PROGRAM EM06_Picking
VAR
	
	//Backbone
	FB_StateMachine_Picking			: FB_StateManager;
	bFl_RunningMachinePicking		: BOOL;
	bFl_SeqReset					: BOOL;
	bFl_Manual						: BOOL;
	CheckStatusPicking				: checkstatus;
	AlarmEventHistory				: ARRAY[1..20] OF Alarm_Event_History;
	ProductFound					: ARRAY [1..4] OF BOOL;
	
	//Motor
	Motor_BoxPicking				: MotorManagement;
	bFl_MotorPicking				: BOOL;
	Motor_Picking_Error				: BOOL;
	Motor_Picking_ErrorID			: UINT;
	
	//Pneumatic
	Pneumatic_GapMaker				: Pneumatic_2Coil_Management;
	bFl_GapMaker_Rtc				: BOOL;
	bFl_GapMaker_Adv				: BOOL;
	Pneu_GapMaker_Error				: BOOL;	
	Pneu_GapMaker_ErrorMsg			: STRING;
	
	Pneumatic_Centering				: Pneumatic_1Coil_Management;
	bFl_Centering					: BOOL;
	Pneu_Centering_Error			: BOOL;	
	Pneu_Centering_ErrorMsg			: STRING;
	
	//Picking
	Picking							: FB_Picking;
	
	//Barcode Reader
	bFl_BarcodeChecked				: BOOL;
	bFl_TriggerBarcode				: BOOL;
	bFl_DoneRead_Barcode_Picking	: ARRAY [1..4] OF BOOL;
	bFl_GoodRead_Barcode_Picking	: ARRAY [1..4] OF BOOL;
	bFl_BadRead_Barcode_Picking		: ARRAY [1..4] OF BOOL;
	BarcodeInspection				: FB_BarcodeInspection;
	BarcodeReader_Picking1			: DM_Connect;
	BarcodeReader_Picking2			: DM_Connect;
	BarcodeReader_Picking3			: DM_Connect;
	BarcodeReader_Picking4			: DM_Connect;
	DataBarcode_Picking1			: STRING;
	DataBarcode_Picking2			: STRING;
	DataBarcode_Picking3			: STRING;
	DataBarcode_Picking4			: STRING;
	Barcode1_Error					: BOOL;
	Barcode2_Error					: BOOL;
	Barcode3_Error					: BOOL;
	Barcode4_Error					: BOOL;
	TestRun							: BOOL;
	TestTrigger						: BOOL;
	LEN1							: INT;
	POS1							: INT;
	POS2							: INT;
	LEN_2							: INT;
	LinkUp							: STRING(255);
	RotatePicking					: RotatePick;
	DonePick						: BOOL;
	bFL_Safety						: BOOL;
	AutoReset						: BOOL;
	TON_Auto						: TON;
	AutoAck							: BOOL;
	AutoRun							: BOOL;
	TOF_Run							: TOF;
	TOF_Reset						: TOF;
	AlarmEventActive				: ARRAY[1..20] OF Alarm_Event_Active;
	RejectMsgList					: RejectMsgHandling;
	bReject							: BOOL;
	RejectID						: INT;
	RejectMsg						: STRING;
	CounterReject					: UINT;
	bRotate							: BOOL;
	BarcodeReader_Picking2B			: DM_Connect;
	Barcode2B_Error					: BOOL;
	DataBarcode_Picking2B			: STRING;
	bFl_DoneRead_Barcode_Picking2B	: BOOL;
	
	BarcodeReader_Picking3B			: DM_Connect;
	Barcode3B_Error					: BOOL;
	DataBarcode_Picking3B			: STRING;
	intRotatePick					: USINT;
END_VAR
VAR // added by the converter: edge detectors and wires of the graphical bodies
    _w1 : BOOL;
END_VAR

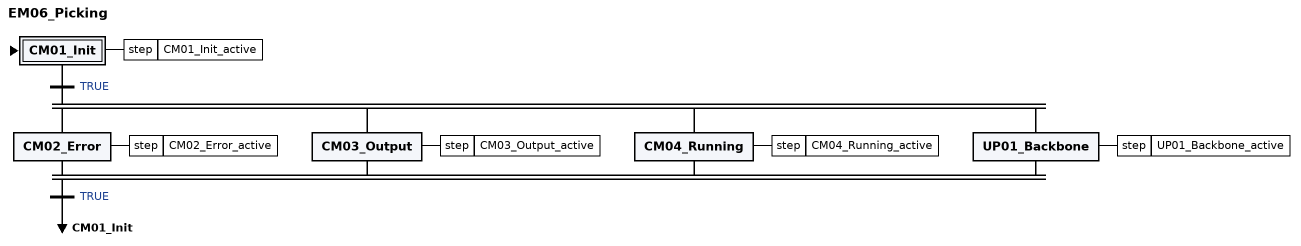
INITIAL_STEP CM01_Init:
    CM01_Init_active(N);  // step action
END_STEP
TRANSITION FROM CM01_Init TO (CM02_Error, CM03_Output, CM04_Running, UP01_Backbone)
    := TRUE;
END_TRANSITION
STEP CM02_Error:
    CM02_Error_active(N);  // step action
END_STEP
STEP CM03_Output:
    CM03_Output_active(N);  // step action
END_STEP
STEP CM04_Running:
    CM04_Running_active(N);  // step action
END_STEP
STEP UP01_Backbone:
    UP01_Backbone_active(N);  // step action
END_STEP
TRANSITION FROM (CM02_Error, CM03_Output, CM04_Running, UP01_Backbone) TO CM01_Init
    := TRUE;
END_TRANSITION

ACTION CM01_Init_active:
Data_GVL.bFL_StartPicking			:= Status_GVL.bFl_RunButton_Robotic OR HMI_GVL.bStartButtonPicking OR HMI_GVL.bAutoStartPicking;
Data_GVL.bFL_StopPicking			:= NOT Status_GVL.bFl_StopButton_Robotic OR HMI_GVL.bStopButtonPicking;
Data_GVL.bFL_ResetPicking			:= Status_GVL.bFl_ResetButton_Robotic OR HMI_GVL.bResetButtonPicking OR HMI_GVL.bAutoResetPicking;
Data_GVL.bFL_AckPicking				:= Status_GVL.bFl_Acknowledge_Robotic OR HMI_GVL.bAcknowledgeButtonPicking OR HMI_GVL.bAutoAcknowledgePicking;
Data_GVL.bFL_AutoManuaModePicking 	:= Status_GVL.bFl_Manual_Robotic OR HMI_GVL.bTestModeEnablePicking;
bFl_RunningMachinePicking			:= Data_GVL.stStateMachinePicking.Running;
bFl_Manual							:= Data_GVL.stStateMachinePicking.ManualMode;
bFl_SeqReset						:= NOT Status_GVL.bFl_EStop_Robotic;
bFL_Safety							:= Status_GVL.bFl_EStop_Robotic AND Status_GVL.bSafety_DoorRobotic AND Status_GVL.bAirPressure_Robotic;



(*=================Convert Timer============================*)
Data_GVL.Tmr_Picking	:= ConvertMilliSecTimeData(HMI_GVL.Tmr_Picking);
Data_GVL.Tmr_Centering	:= ConvertMilliSecTimeData(HMI_GVL.Tmr_Centering);

(*=================Auto Flushing============================*)
//Place1
IF ProductFound[1] AND HMI_GVL.arCountReal[1] > 1 THEN
	Status_GVL.AutoFlush_Placing1	:= TRUE;
ELSE
	Status_GVL.AutoFlush_Placing1	:= FALSE;
END_IF

//Place2
IF ProductFound[2] AND HMI_GVL.arCountReal[2] > 1 THEN
	Status_GVL.AutoFlush_Placing2	:= TRUE;
ELSE
	Status_GVL.AutoFlush_Placing2	:= FALSE;
END_IF

//Place3
IF ProductFound[3] AND HMI_GVL.arCountReal[3] > 1 THEN
	Status_GVL.AutoFlush_Placing3	:= TRUE;
ELSE
	Status_GVL.AutoFlush_Placing3	:= FALSE;
END_IF

//Place4
IF ProductFound[4] AND HMI_GVL.arCountReal[4] > 1 THEN
	Status_GVL.AutoFlush_Placing4	:= TRUE;
ELSE
	Status_GVL.AutoFlush_Placing4	:= FALSE;
END_IF
END_ACTION

ACTION CM02_Error_active:
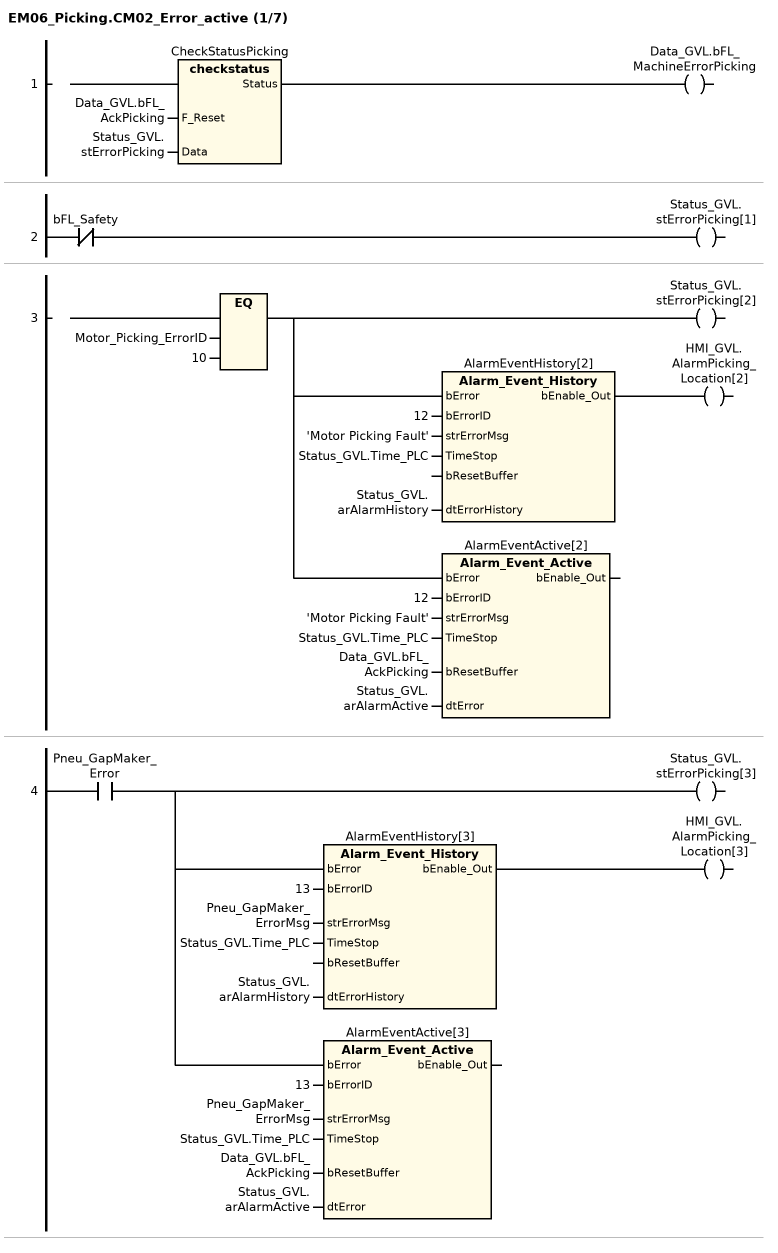
// NETWORK 1
CheckStatusPicking(F_Reset := Data_GVL.bFL_AckPicking, Data := Status_GVL.stErrorPicking); // checkstatus
Data_GVL.bFL_MachineErrorPicking := CheckStatusPicking.Status;

// NETWORK 2
Status_GVL.stErrorPicking[1] := NOT bFL_Safety;

// NETWORK 3
_w1 := Motor_Picking_ErrorID = 10;
Status_GVL.stErrorPicking[2] := _w1;
AlarmEventHistory[2](
    bError := _w1,
    bErrorID := 12,
    strErrorMsg := 'Motor Picking Fault',
    TimeStop := Status_GVL.Time_PLC,
    dtErrorHistory := Status_GVL.arAlarmHistory); // Alarm_Event_History
HMI_GVL.AlarmPicking_Location[2] := AlarmEventHistory[2].bEnable_Out;
AlarmEventActive[2](
    bError := _w1,
    bErrorID := 12,
    strErrorMsg := 'Motor Picking Fault',
    TimeStop := Status_GVL.Time_PLC,
    bResetBuffer := Data_GVL.bFL_AckPicking,
    dtError := Status_GVL.arAlarmActive); // Alarm_Event_Active

// NETWORK 4
Status_GVL.stErrorPicking[3] := Pneu_GapMaker_Error;
AlarmEventHistory[3](
    bError := Pneu_GapMaker_Error,
    bErrorID := 13,
    strErrorMsg := Pneu_GapMaker_ErrorMsg,
    TimeStop := Status_GVL.Time_PLC,
    dtErrorHistory := Status_GVL.arAlarmHistory); // Alarm_Event_History
HMI_GVL.AlarmPicking_Location[3] := AlarmEventHistory[3].bEnable_Out;
AlarmEventActive[3](
    bError := Pneu_GapMaker_Error,
    bErrorID := 13,
    strErrorMsg := Pneu_GapMaker_ErrorMsg,
    TimeStop := Status_GVL.Time_PLC,
    bResetBuffer := Data_GVL.bFL_AckPicking,
    dtError := Status_GVL.arAlarmActive); // Alarm_Event_Active

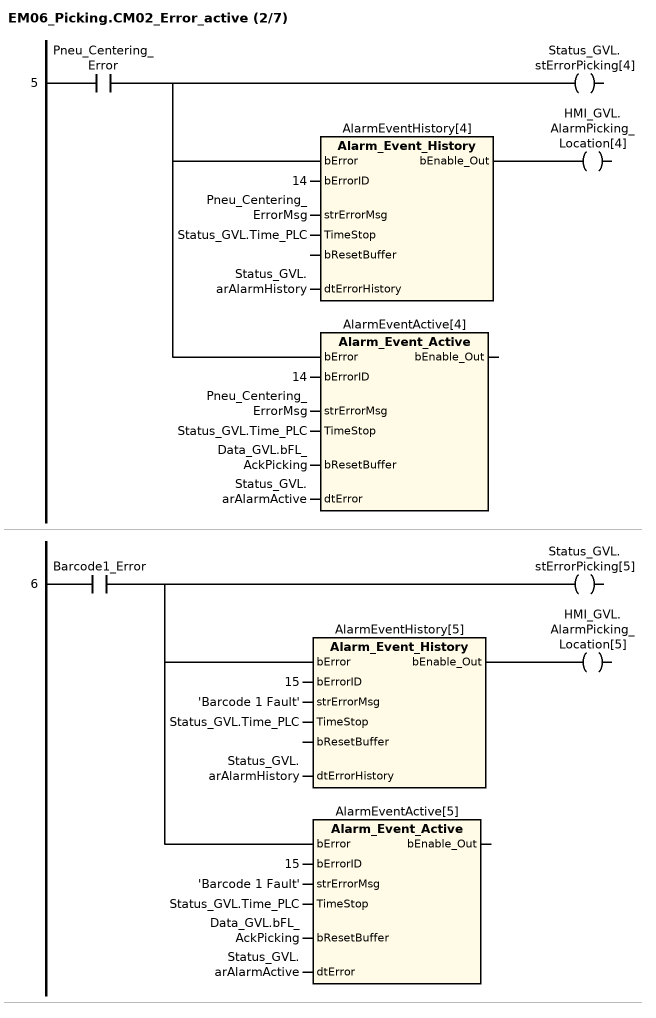
// NETWORK 5
Status_GVL.stErrorPicking[4] := Pneu_Centering_Error;
AlarmEventHistory[4](
    bError := Pneu_Centering_Error,
    bErrorID := 14,
    strErrorMsg := Pneu_Centering_ErrorMsg,
    TimeStop := Status_GVL.Time_PLC,
    dtErrorHistory := Status_GVL.arAlarmHistory); // Alarm_Event_History
HMI_GVL.AlarmPicking_Location[4] := AlarmEventHistory[4].bEnable_Out;
AlarmEventActive[4](
    bError := Pneu_Centering_Error,
    bErrorID := 14,
    strErrorMsg := Pneu_Centering_ErrorMsg,
    TimeStop := Status_GVL.Time_PLC,
    bResetBuffer := Data_GVL.bFL_AckPicking,
    dtError := Status_GVL.arAlarmActive); // Alarm_Event_Active

// NETWORK 6
Status_GVL.stErrorPicking[5] := Barcode1_Error;
AlarmEventHistory[5](
    bError := Barcode1_Error,
    bErrorID := 15,
    strErrorMsg := 'Barcode 1 Fault',
    TimeStop := Status_GVL.Time_PLC,
    dtErrorHistory := Status_GVL.arAlarmHistory); // Alarm_Event_History
HMI_GVL.AlarmPicking_Location[5] := AlarmEventHistory[5].bEnable_Out;
AlarmEventActive[5](
    bError := Barcode1_Error,
    bErrorID := 15,
    strErrorMsg := 'Barcode 1 Fault',
    TimeStop := Status_GVL.Time_PLC,
    bResetBuffer := Data_GVL.bFL_AckPicking,
    dtError := Status_GVL.arAlarmActive); // Alarm_Event_Active

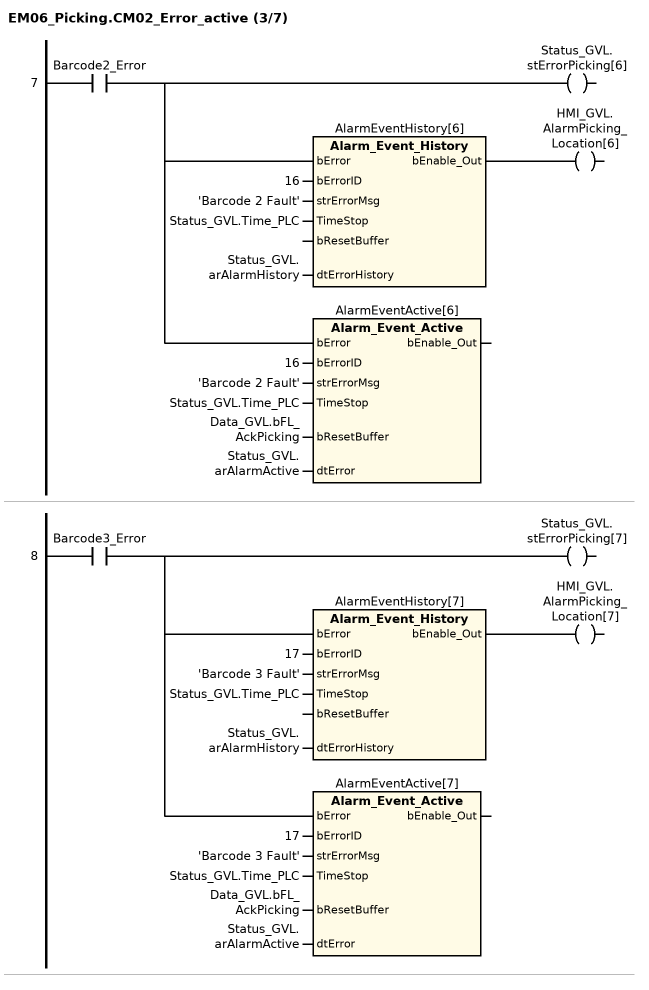
// NETWORK 7
Status_GVL.stErrorPicking[6] := Barcode2_Error;
AlarmEventHistory[6](
    bError := Barcode2_Error,
    bErrorID := 16,
    strErrorMsg := 'Barcode 2 Fault',
    TimeStop := Status_GVL.Time_PLC,
    dtErrorHistory := Status_GVL.arAlarmHistory); // Alarm_Event_History
HMI_GVL.AlarmPicking_Location[6] := AlarmEventHistory[6].bEnable_Out;
AlarmEventActive[6](
    bError := Barcode2_Error,
    bErrorID := 16,
    strErrorMsg := 'Barcode 2 Fault',
    TimeStop := Status_GVL.Time_PLC,
    bResetBuffer := Data_GVL.bFL_AckPicking,
    dtError := Status_GVL.arAlarmActive); // Alarm_Event_Active

// NETWORK 8
Status_GVL.stErrorPicking[7] := Barcode3_Error;
AlarmEventHistory[7](
    bError := Barcode3_Error,
    bErrorID := 17,
    strErrorMsg := 'Barcode 3 Fault',
    TimeStop := Status_GVL.Time_PLC,
    dtErrorHistory := Status_GVL.arAlarmHistory); // Alarm_Event_History
HMI_GVL.AlarmPicking_Location[7] := AlarmEventHistory[7].bEnable_Out;
AlarmEventActive[7](
    bError := Barcode3_Error,
    bErrorID := 17,
    strErrorMsg := 'Barcode 3 Fault',
    TimeStop := Status_GVL.Time_PLC,
    bResetBuffer := Data_GVL.bFL_AckPicking,
    dtError := Status_GVL.arAlarmActive); // Alarm_Event_Active

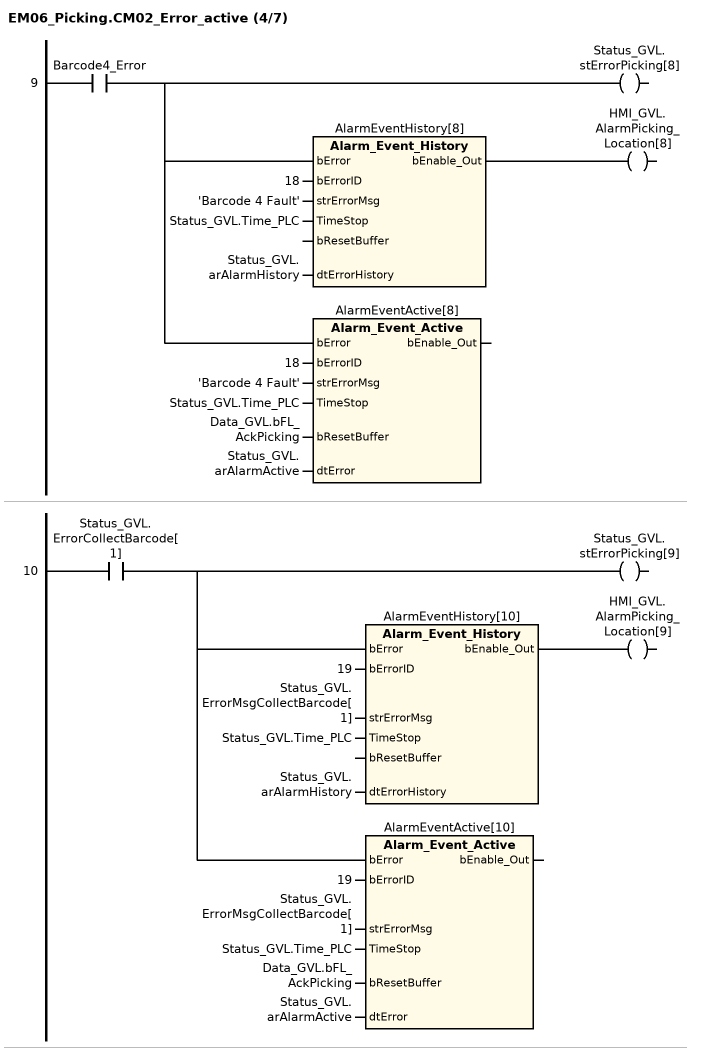
// NETWORK 9
Status_GVL.stErrorPicking[8] := Barcode4_Error;
AlarmEventHistory[8](
    bError := Barcode4_Error,
    bErrorID := 18,
    strErrorMsg := 'Barcode 4 Fault',
    TimeStop := Status_GVL.Time_PLC,
    dtErrorHistory := Status_GVL.arAlarmHistory); // Alarm_Event_History
HMI_GVL.AlarmPicking_Location[8] := AlarmEventHistory[8].bEnable_Out;
AlarmEventActive[8](
    bError := Barcode4_Error,
    bErrorID := 18,
    strErrorMsg := 'Barcode 4 Fault',
    TimeStop := Status_GVL.Time_PLC,
    bResetBuffer := Data_GVL.bFL_AckPicking,
    dtError := Status_GVL.arAlarmActive); // Alarm_Event_Active

// NETWORK 10
Status_GVL.stErrorPicking[9] := Status_GVL.ErrorCollectBarcode[1];
AlarmEventHistory[10](
    bError := Status_GVL.ErrorCollectBarcode[1],
    bErrorID := 19,
    strErrorMsg := Status_GVL.ErrorMsgCollectBarcode[1],
    TimeStop := Status_GVL.Time_PLC,
    dtErrorHistory := Status_GVL.arAlarmHistory); // Alarm_Event_History
HMI_GVL.AlarmPicking_Location[9] := AlarmEventHistory[10].bEnable_Out;
AlarmEventActive[10](
    bError := Status_GVL.ErrorCollectBarcode[1],
    bErrorID := 19,
    strErrorMsg := Status_GVL.ErrorMsgCollectBarcode[1],
    TimeStop := Status_GVL.Time_PLC,
    bResetBuffer := Data_GVL.bFL_AckPicking,
    dtError := Status_GVL.arAlarmActive); // Alarm_Event_Active

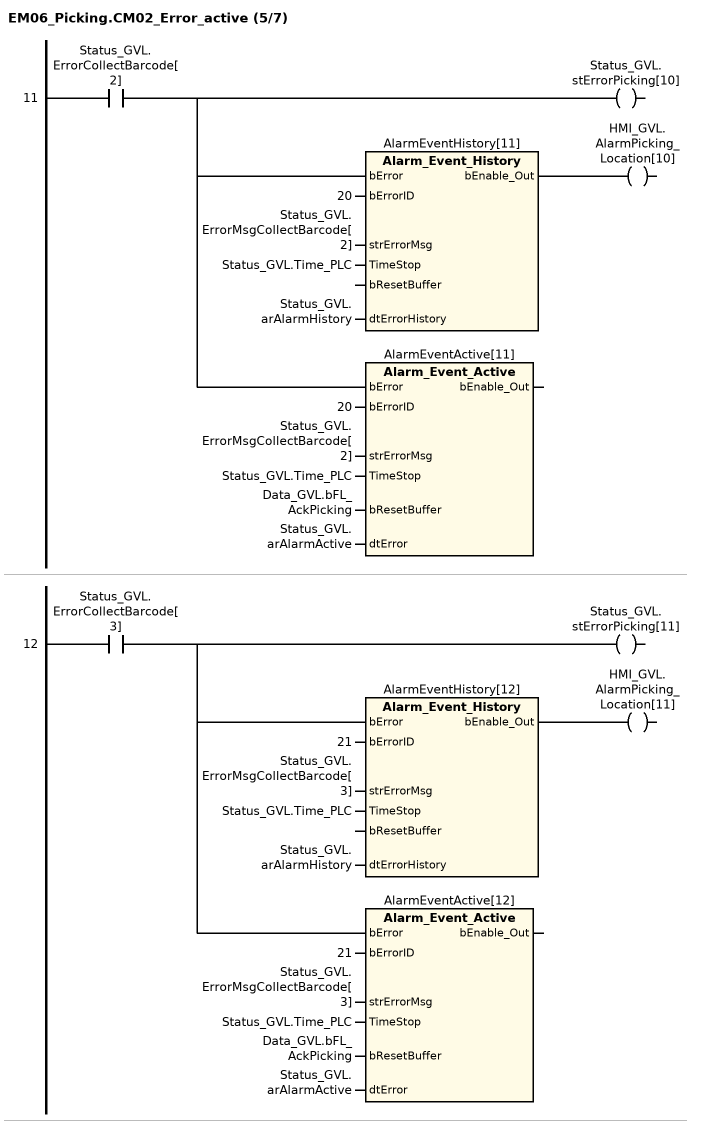
// NETWORK 11
Status_GVL.stErrorPicking[10] := Status_GVL.ErrorCollectBarcode[2];
AlarmEventHistory[11](
    bError := Status_GVL.ErrorCollectBarcode[2],
    bErrorID := 20,
    strErrorMsg := Status_GVL.ErrorMsgCollectBarcode[2],
    TimeStop := Status_GVL.Time_PLC,
    dtErrorHistory := Status_GVL.arAlarmHistory); // Alarm_Event_History
HMI_GVL.AlarmPicking_Location[10] := AlarmEventHistory[11].bEnable_Out;
AlarmEventActive[11](
    bError := Status_GVL.ErrorCollectBarcode[2],
    bErrorID := 20,
    strErrorMsg := Status_GVL.ErrorMsgCollectBarcode[2],
    TimeStop := Status_GVL.Time_PLC,
    bResetBuffer := Data_GVL.bFL_AckPicking,
    dtError := Status_GVL.arAlarmActive); // Alarm_Event_Active

// NETWORK 12
Status_GVL.stErrorPicking[11] := Status_GVL.ErrorCollectBarcode[3];
AlarmEventHistory[12](
    bError := Status_GVL.ErrorCollectBarcode[3],
    bErrorID := 21,
    strErrorMsg := Status_GVL.ErrorMsgCollectBarcode[3],
    TimeStop := Status_GVL.Time_PLC,
    dtErrorHistory := Status_GVL.arAlarmHistory); // Alarm_Event_History
HMI_GVL.AlarmPicking_Location[11] := AlarmEventHistory[12].bEnable_Out;
AlarmEventActive[12](
    bError := Status_GVL.ErrorCollectBarcode[3],
    bErrorID := 21,
    strErrorMsg := Status_GVL.ErrorMsgCollectBarcode[3],
    TimeStop := Status_GVL.Time_PLC,
    bResetBuffer := Data_GVL.bFL_AckPicking,
    dtError := Status_GVL.arAlarmActive); // Alarm_Event_Active

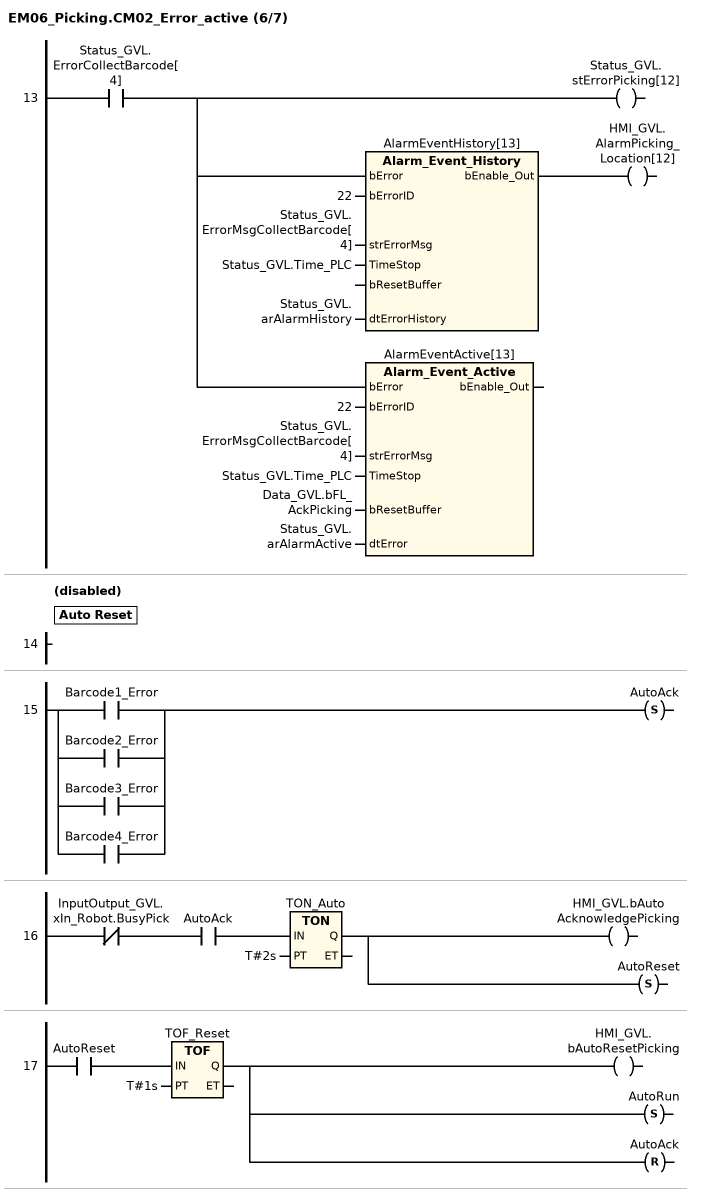
// NETWORK 13
Status_GVL.stErrorPicking[12] := Status_GVL.ErrorCollectBarcode[4];
AlarmEventHistory[13](
    bError := Status_GVL.ErrorCollectBarcode[4],
    bErrorID := 22,
    strErrorMsg := Status_GVL.ErrorMsgCollectBarcode[4],
    TimeStop := Status_GVL.Time_PLC,
    dtErrorHistory := Status_GVL.arAlarmHistory); // Alarm_Event_History
HMI_GVL.AlarmPicking_Location[12] := AlarmEventHistory[13].bEnable_Out;
AlarmEventActive[13](
    bError := Status_GVL.ErrorCollectBarcode[4],
    bErrorID := 22,
    strErrorMsg := Status_GVL.ErrorMsgCollectBarcode[4],
    TimeStop := Status_GVL.Time_PLC,
    bResetBuffer := Data_GVL.bFL_AckPicking,
    dtError := Status_GVL.arAlarmActive); // Alarm_Event_Active

// NETWORK 14 (disabled)
// label: Auto Reset

// NETWORK 15
AutoAck S= Barcode1_Error OR Barcode2_Error OR Barcode3_Error OR Barcode4_Error;

// NETWORK 16
TON_Auto(IN := NOT InputOutput_GVL.xIn_Robot.BusyPick AND AutoAck, PT := T#2s); // TON
HMI_GVL.bAutoAcknowledgePicking := TON_Auto.Q;
AutoReset S= TON_Auto.Q;

// NETWORK 17
TOF_Reset(IN := AutoReset, PT := T#1s); // TOF
HMI_GVL.bAutoResetPicking := TOF_Reset.Q;
AutoRun S= TOF_Reset.Q;
AutoAck R= TOF_Reset.Q;

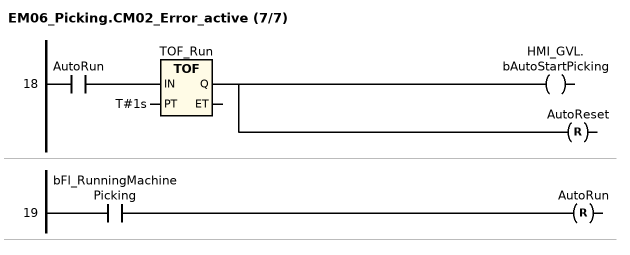
// NETWORK 18
TOF_Run(IN := AutoRun, PT := T#1s); // TOF
HMI_GVL.bAutoStartPicking := TOF_Run.Q;
AutoReset R= TOF_Run.Q;

// NETWORK 19
AutoRun R= bFl_RunningMachinePicking;
END_ACTION

ACTION CM03_Output_active:
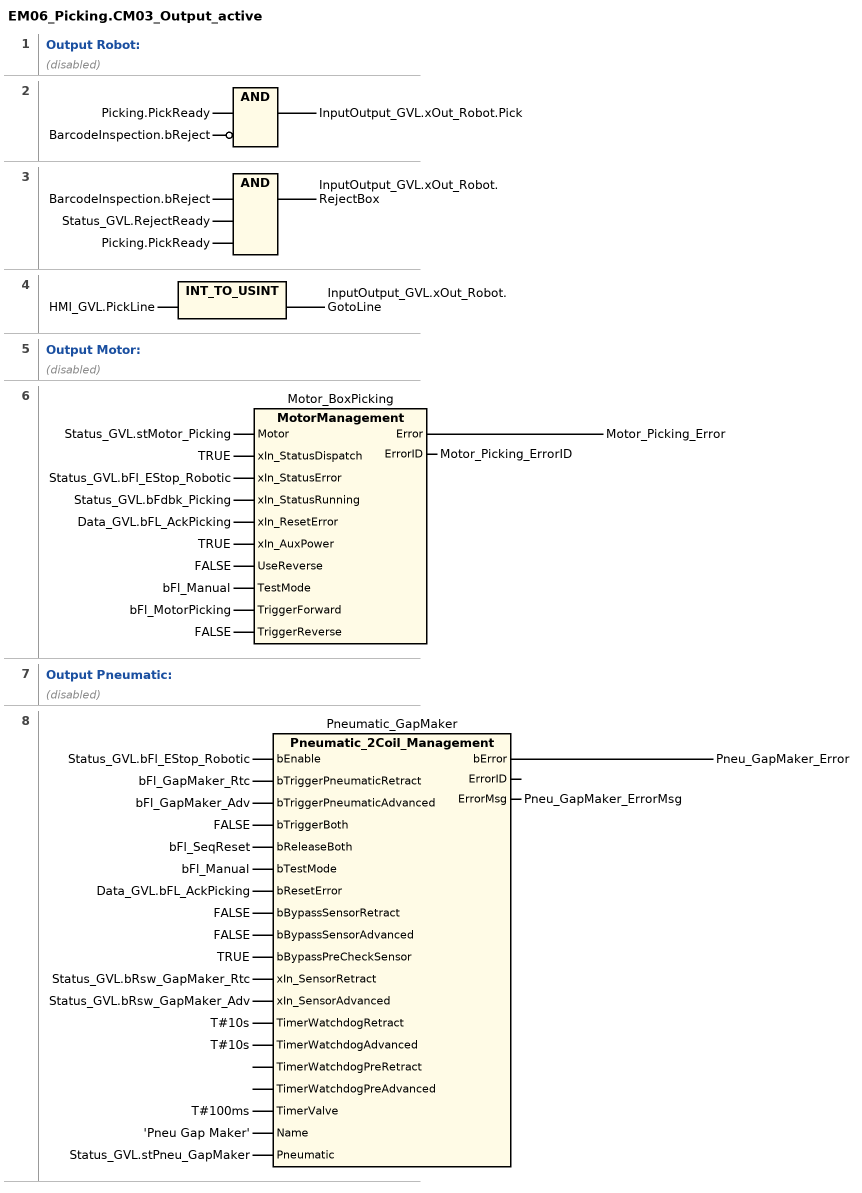
// NETWORK 1 (disabled)
// label: Output Robot

// NETWORK 2
InputOutput_GVL.xOut_Robot.Pick := Picking.PickReady AND NOT BarcodeInspection.bReject;

// NETWORK 3
InputOutput_GVL.xOut_Robot.RejectBox := BarcodeInspection.bReject AND Status_GVL.RejectReady AND Picking.PickReady;

// NETWORK 4
InputOutput_GVL.xOut_Robot.GotoLine := INT_TO_USINT(HMI_GVL.PickLine);

// NETWORK 5 (disabled)
// label: Output Motor

// NETWORK 6
Motor_BoxPicking(
    Motor := Status_GVL.stMotor_Picking,
    xIn_StatusDispatch := TRUE,
    xIn_StatusError := Status_GVL.bFl_EStop_Robotic,
    xIn_StatusRunning := Status_GVL.bFdbk_Picking,
    xIn_ResetError := Data_GVL.bFL_AckPicking,
    xIn_AuxPower := TRUE,
    UseReverse := FALSE,
    TestMode := bFl_Manual,
    TriggerForward := bFl_MotorPicking,
    TriggerReverse := FALSE,
    ErrorID => Motor_Picking_ErrorID); // MotorManagement
Motor_Picking_Error := Motor_BoxPicking.Error;

// NETWORK 7 (disabled)
// label: Output Pneumatic

// NETWORK 8
Pneumatic_GapMaker(
    bEnable := Status_GVL.bFl_EStop_Robotic,
    bTriggerPneumaticRetract := bFl_GapMaker_Rtc,
    bTriggerPneumaticAdvanced := bFl_GapMaker_Adv,
    bTriggerBoth := FALSE,
    bReleaseBoth := bFl_SeqReset,
    bTestMode := bFl_Manual,
    bResetError := Data_GVL.bFL_AckPicking,
    bBypassSensorRetract := FALSE,
    bBypassSensorAdvanced := FALSE,
    bBypassPreCheckSensor := TRUE,
    xIn_SensorRetract := Status_GVL.bRsw_GapMaker_Rtc,
    xIn_SensorAdvanced := Status_GVL.bRsw_GapMaker_Adv,
    TimerWatchdogRetract := T#10s,
    TimerWatchdogAdvanced := T#10s,
    TimerValve := T#100ms,
    Name := 'Pneu Gap Maker',
    Pneumatic := Status_GVL.stPneu_GapMaker,
    ErrorMsg => Pneu_GapMaker_ErrorMsg); // Pneumatic_2Coil_Management
Pneu_GapMaker_Error := Pneumatic_GapMaker.bError;

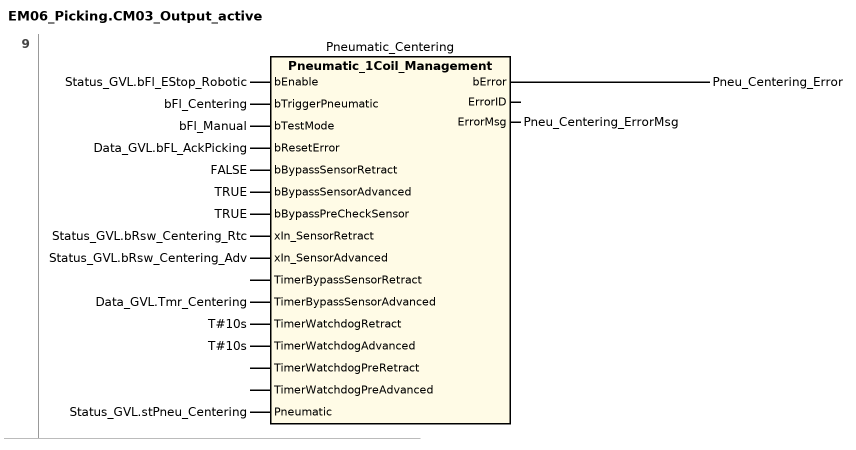
// NETWORK 9
Pneumatic_Centering(
    bEnable := Status_GVL.bFl_EStop_Robotic,
    bTriggerPneumatic := bFl_Centering,
    bTestMode := bFl_Manual,
    bResetError := Data_GVL.bFL_AckPicking,
    bBypassSensorRetract := FALSE,
    bBypassSensorAdvanced := TRUE,
    bBypassPreCheckSensor := TRUE,
    xIn_SensorRetract := Status_GVL.bRsw_Centering_Rtc,
    xIn_SensorAdvanced := Status_GVL.bRsw_Centering_Adv,
    TimerBypassSensorAdvanced := Data_GVL.Tmr_Centering,
    TimerWatchdogRetract := T#10s,
    TimerWatchdogAdvanced := T#10s,
    Pneumatic := Status_GVL.stPneu_Centering,
    ErrorMsg => Pneu_Centering_ErrorMsg); // Pneumatic_1Coil_Management
Pneu_Centering_Error := Pneumatic_Centering.bError;
END_ACTION

ACTION CM04_Running_active:
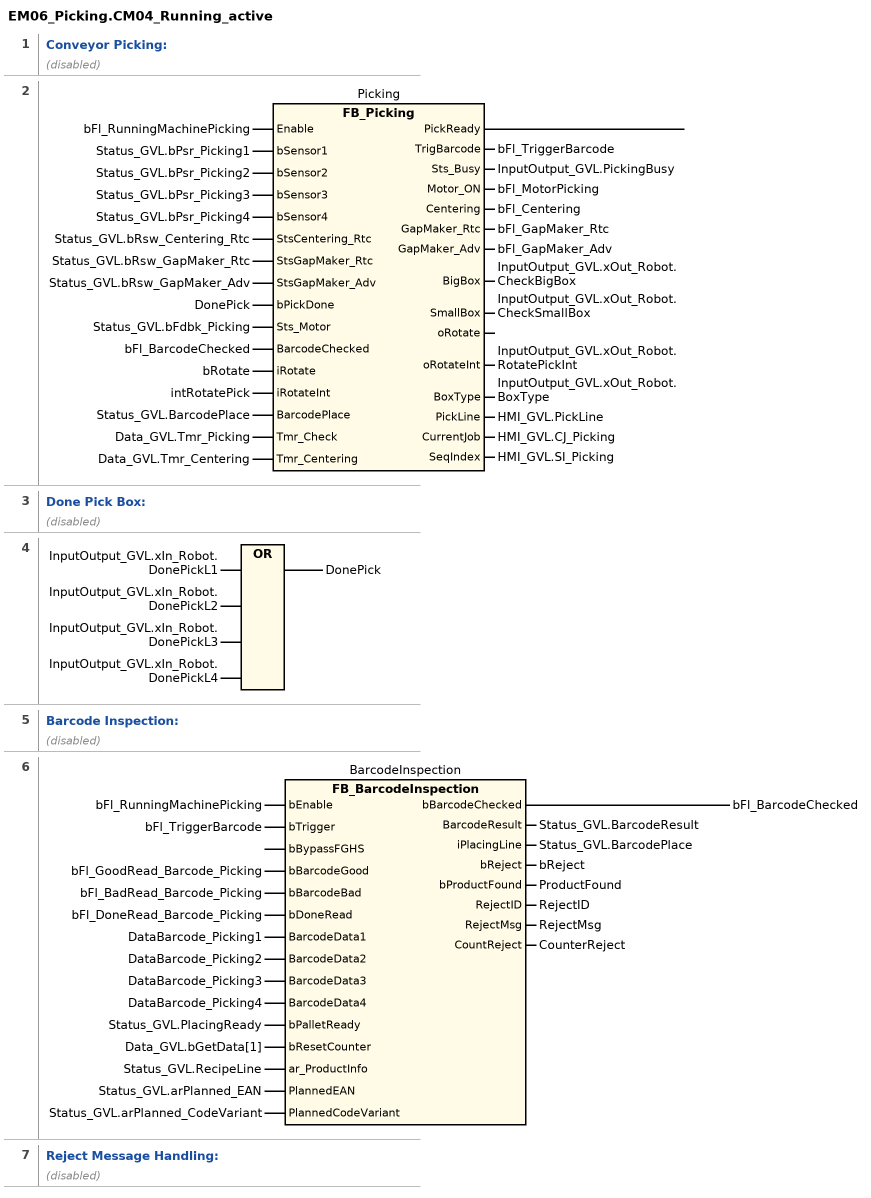
// NETWORK 1 (disabled)
// label: Conveyor Picking

// NETWORK 2
Picking(
    Enable := bFl_RunningMachinePicking,
    bSensor1 := Status_GVL.bPsr_Picking1,
    bSensor2 := Status_GVL.bPsr_Picking2,
    bSensor3 := Status_GVL.bPsr_Picking3,
    bSensor4 := Status_GVL.bPsr_Picking4,
    StsCentering_Rtc := Status_GVL.bRsw_Centering_Rtc,
    StsGapMaker_Rtc := Status_GVL.bRsw_GapMaker_Rtc,
    StsGapMaker_Adv := Status_GVL.bRsw_GapMaker_Adv,
    bPickDone := DonePick,
    Sts_Motor := Status_GVL.bFdbk_Picking,
    BarcodeChecked := bFl_BarcodeChecked,
    iRotate := bRotate,
    iRotateInt := intRotatePick,
    BarcodePlace := Status_GVL.BarcodePlace,
    Tmr_Check := Data_GVL.Tmr_Picking,
    Tmr_Centering := Data_GVL.Tmr_Centering,
    TrigBarcode => bFl_TriggerBarcode,
    Sts_Busy => InputOutput_GVL.PickingBusy,
    Motor_ON => bFl_MotorPicking,
    Centering => bFl_Centering,
    GapMaker_Rtc => bFl_GapMaker_Rtc,
    GapMaker_Adv => bFl_GapMaker_Adv,
    BigBox => InputOutput_GVL.xOut_Robot.CheckBigBox,
    SmallBox => InputOutput_GVL.xOut_Robot.CheckSmallBox,
    oRotateInt => InputOutput_GVL.xOut_Robot.RotatePickInt,
    BoxType => InputOutput_GVL.xOut_Robot.BoxType,
    PickLine => HMI_GVL.PickLine,
    CurrentJob => HMI_GVL.CJ_Picking,
    SeqIndex => HMI_GVL.SI_Picking); // FB_Picking

// NETWORK 3 (disabled)
// label: Done Pick Box

// NETWORK 4
DonePick := InputOutput_GVL.xIn_Robot.DonePickL1 OR InputOutput_GVL.xIn_Robot.DonePickL2 OR InputOutput_GVL.xIn_Robot.DonePickL3 OR InputOutput_GVL.xIn_Robot.DonePickL4;

// NETWORK 5 (disabled)
// label: Barcode Inspection

// NETWORK 6
BarcodeInspection(
    bEnable := bFl_RunningMachinePicking,
    bTrigger := bFl_TriggerBarcode,
    bBarcodeGood := bFl_GoodRead_Barcode_Picking,
    bBarcodeBad := bFl_BadRead_Barcode_Picking,
    bDoneRead := bFl_DoneRead_Barcode_Picking,
    BarcodeData1 := DataBarcode_Picking1,
    BarcodeData2 := DataBarcode_Picking2,
    BarcodeData3 := DataBarcode_Picking3,
    BarcodeData4 := DataBarcode_Picking4,
    bPalletReady := Status_GVL.PlacingReady,
    bResetCounter := Data_GVL.bGetData[1],
    ar_ProductInfo := Status_GVL.RecipeLine,
    PlannedEAN := Status_GVL.arPlanned_EAN,
    PlannedCodeVariant := Status_GVL.arPlanned_CodeVariant,
    BarcodeResult => Status_GVL.BarcodeResult,
    iPlacingLine => Status_GVL.BarcodePlace,
    bReject => bReject,
    bProductFound => ProductFound,
    RejectID => RejectID,
    RejectMsg => RejectMsg,
    CountReject => CounterReject); // FB_BarcodeInspection
bFl_BarcodeChecked := BarcodeInspection.bBarcodeChecked;

// NETWORK 7 (disabled)
// label: Reject Message Handling

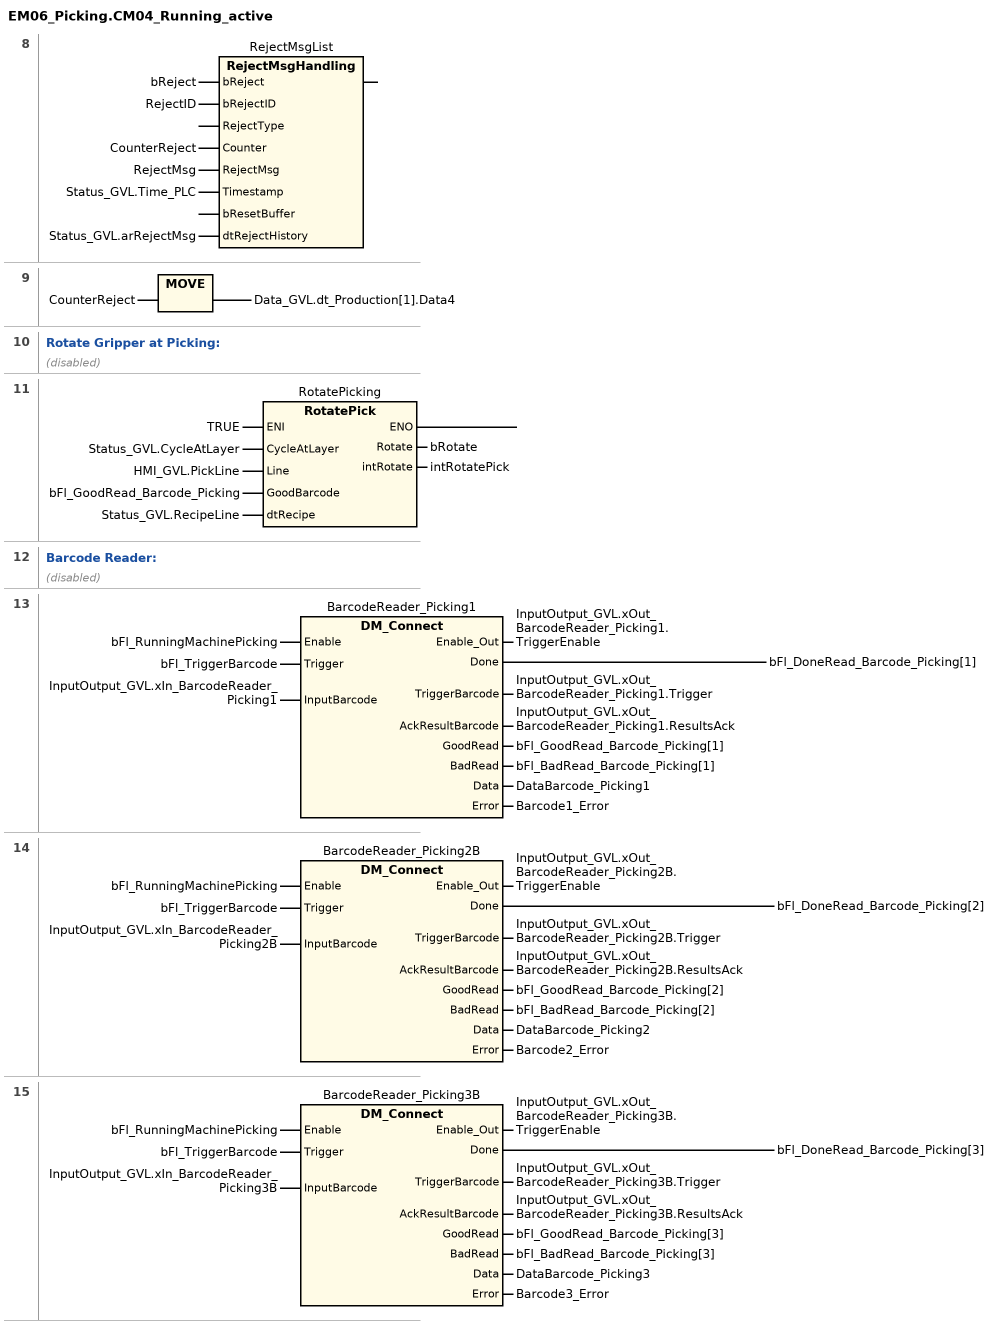
// NETWORK 8
RejectMsgList(
    bReject := bReject,
    bRejectID := RejectID,
    Counter := CounterReject,
    RejectMsg := RejectMsg,
    Timestamp := Status_GVL.Time_PLC,
    dtRejectHistory := Status_GVL.arRejectMsg); // RejectMsgHandling

// NETWORK 9
Data_GVL.dt_Production[1].Data4 := CounterReject;

// NETWORK 10 (disabled)
// label: Rotate Gripper at Picking

// NETWORK 11
RotatePicking(
    ENI := TRUE,
    CycleAtLayer := Status_GVL.CycleAtLayer,
    Line := HMI_GVL.PickLine,
    GoodBarcode := bFl_GoodRead_Barcode_Picking,
    dtRecipe := Status_GVL.RecipeLine,
    Rotate => bRotate,
    intRotate => intRotatePick); // RotatePick

// NETWORK 12 (disabled)
// label: Barcode Reader

// NETWORK 13
BarcodeReader_Picking1(
    Enable := bFl_RunningMachinePicking,
    Trigger := bFl_TriggerBarcode,
    InputBarcode := InputOutput_GVL.xIn_BarcodeReader_Picking1,
    Enable_Out => InputOutput_GVL.xOut_BarcodeReader_Picking1.TriggerEnable,
    TriggerBarcode => InputOutput_GVL.xOut_BarcodeReader_Picking1.Trigger,
    AckResultBarcode => InputOutput_GVL.xOut_BarcodeReader_Picking1.ResultsAck,
    GoodRead => bFl_GoodRead_Barcode_Picking[1],
    BadRead => bFl_BadRead_Barcode_Picking[1],
    Data => DataBarcode_Picking1,
    Error => Barcode1_Error); // DM_Connect
bFl_DoneRead_Barcode_Picking[1] := BarcodeReader_Picking1.Done;

// NETWORK 14
BarcodeReader_Picking2B(
    Enable := bFl_RunningMachinePicking,
    Trigger := bFl_TriggerBarcode,
    InputBarcode := InputOutput_GVL.xIn_BarcodeReader_Picking2B,
    Enable_Out => InputOutput_GVL.xOut_BarcodeReader_Picking2B.TriggerEnable,
    TriggerBarcode => InputOutput_GVL.xOut_BarcodeReader_Picking2B.Trigger,
    AckResultBarcode => InputOutput_GVL.xOut_BarcodeReader_Picking2B.ResultsAck,
    GoodRead => bFl_GoodRead_Barcode_Picking[2],
    BadRead => bFl_BadRead_Barcode_Picking[2],
    Data => DataBarcode_Picking2,
    Error => Barcode2_Error); // DM_Connect
bFl_DoneRead_Barcode_Picking[2] := BarcodeReader_Picking2B.Done;

// NETWORK 15
BarcodeReader_Picking3B(
    Enable := bFl_RunningMachinePicking,
    Trigger := bFl_TriggerBarcode,
    InputBarcode := InputOutput_GVL.xIn_BarcodeReader_Picking3B,
    Enable_Out => InputOutput_GVL.xOut_BarcodeReader_Picking3B.TriggerEnable,
    TriggerBarcode => InputOutput_GVL.xOut_BarcodeReader_Picking3B.Trigger,
    AckResultBarcode => InputOutput_GVL.xOut_BarcodeReader_Picking3B.ResultsAck,
    GoodRead => bFl_GoodRead_Barcode_Picking[3],
    BadRead => bFl_BadRead_Barcode_Picking[3],
    Data => DataBarcode_Picking3,
    Error => Barcode3_Error); // DM_Connect
bFl_DoneRead_Barcode_Picking[3] := BarcodeReader_Picking3B.Done;

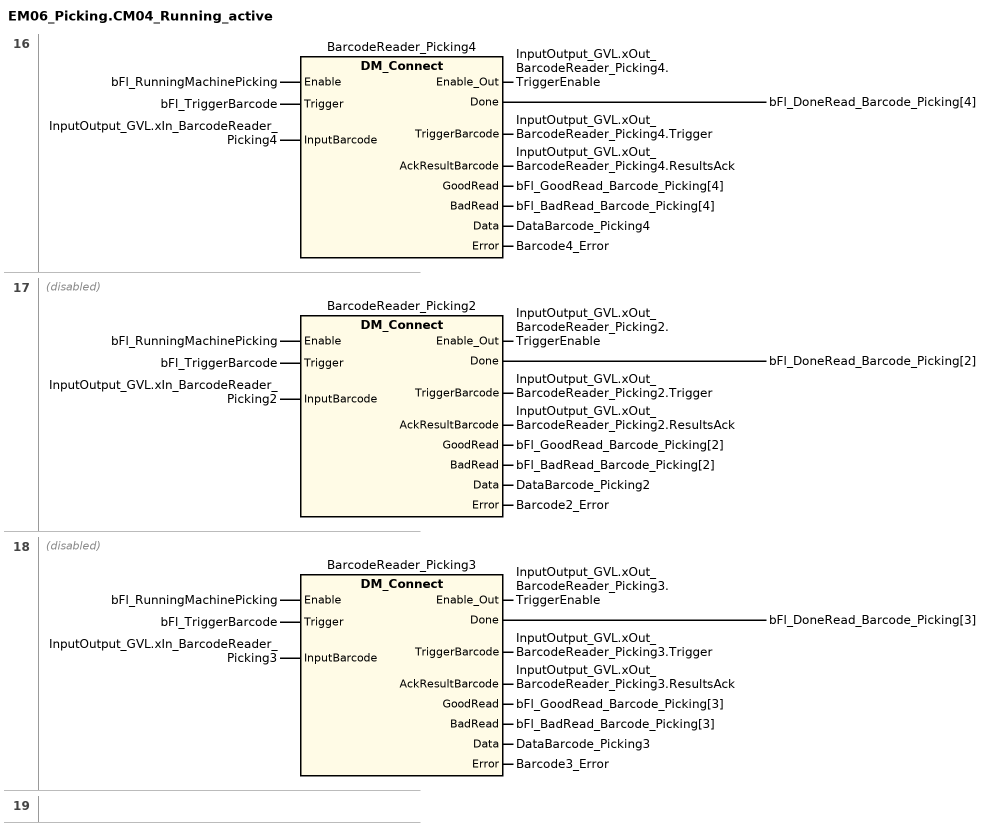
// NETWORK 16
BarcodeReader_Picking4(
    Enable := bFl_RunningMachinePicking,
    Trigger := bFl_TriggerBarcode,
    InputBarcode := InputOutput_GVL.xIn_BarcodeReader_Picking4,
    Enable_Out => InputOutput_GVL.xOut_BarcodeReader_Picking4.TriggerEnable,
    TriggerBarcode => InputOutput_GVL.xOut_BarcodeReader_Picking4.Trigger,
    AckResultBarcode => InputOutput_GVL.xOut_BarcodeReader_Picking4.ResultsAck,
    GoodRead => bFl_GoodRead_Barcode_Picking[4],
    BadRead => bFl_BadRead_Barcode_Picking[4],
    Data => DataBarcode_Picking4,
    Error => Barcode4_Error); // DM_Connect
bFl_DoneRead_Barcode_Picking[4] := BarcodeReader_Picking4.Done;

// NETWORK 17 (disabled)
// BarcodeReader_Picking2(
//     Enable := bFl_RunningMachinePicking,
//     Trigger := bFl_TriggerBarcode,
//     InputBarcode := InputOutput_GVL.xIn_BarcodeReader_Picking2,
//     Enable_Out => InputOutput_GVL.xOut_BarcodeReader_Picking2.TriggerEnable,
//     TriggerBarcode => InputOutput_GVL.xOut_BarcodeReader_Picking2.Trigger,
//     AckResultBarcode => InputOutput_GVL.xOut_BarcodeReader_Picking2.ResultsAck,
//     GoodRead => bFl_GoodRead_Barcode_Picking[2],
//     BadRead => bFl_BadRead_Barcode_Picking[2],
//     Data => DataBarcode_Picking2,
//     Error => Barcode2_Error); // DM_Connect
// bFl_DoneRead_Barcode_Picking[2] := BarcodeReader_Picking2.Done;

// NETWORK 18 (disabled)
// BarcodeReader_Picking3(
//     Enable := bFl_RunningMachinePicking,
//     Trigger := bFl_TriggerBarcode,
//     InputBarcode := InputOutput_GVL.xIn_BarcodeReader_Picking3,
//     Enable_Out => InputOutput_GVL.xOut_BarcodeReader_Picking3.TriggerEnable,
//     TriggerBarcode => InputOutput_GVL.xOut_BarcodeReader_Picking3.Trigger,
//     AckResultBarcode => InputOutput_GVL.xOut_BarcodeReader_Picking3.ResultsAck,
//     GoodRead => bFl_GoodRead_Barcode_Picking[3],
//     BadRead => bFl_BadRead_Barcode_Picking[3],
//     Data => DataBarcode_Picking3,
//     Error => Barcode3_Error); // DM_Connect
// bFl_DoneRead_Barcode_Picking[3] := BarcodeReader_Picking3.Done;

// NETWORK 19
END_ACTION

ACTION UP01_Backbone_active:
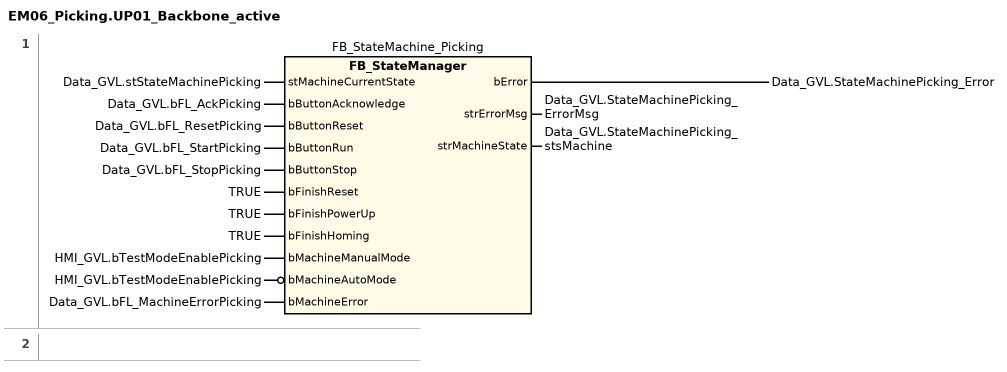
// NETWORK 1
FB_StateMachine_Picking(
    stMachineCurrentState := Data_GVL.stStateMachinePicking,
    bButtonAcknowledge := Data_GVL.bFL_AckPicking,
    bButtonReset := Data_GVL.bFL_ResetPicking,
    bButtonRun := Data_GVL.bFL_StartPicking,
    bButtonStop := Data_GVL.bFL_StopPicking,
    bFinishReset := TRUE,
    bFinishPowerUp := TRUE,
    bFinishHoming := TRUE,
    bMachineManualMode := HMI_GVL.bTestModeEnablePicking,
    bMachineAutoMode := NOT HMI_GVL.bTestModeEnablePicking,
    bMachineError := Data_GVL.bFL_MachineErrorPicking,
    strErrorMsg => Data_GVL.StateMachinePicking_ErrorMsg,
    strMachineState => Data_GVL.StateMachinePicking_stsMachine); // FB_StateManager
Data_GVL.StateMachinePicking_Error := FB_StateMachine_Picking.bError;

// NETWORK 2
END_ACTION

END_PROGRAM

(* stored: Version 1.1.0.1, ProductVersion 3.1.4024.12
   POU EM06_Picking: Id {54c1868d-c4e5-4034-8ce2-3f1edf6df466}, SpecialFunc None
   Action CM01_Init_active: Id {d322bd20-a948-4c0c-888a-00796aebe03a}
   Action CM02_Error_active: Id {19fd0aad-b82a-4ca4-97ab-ee59d8fb8857}
   Action CM03_Output_active: Id {9cd97ce9-65cb-4914-9788-e6c3cfab2498}
   Action CM04_Running_active: Id {7494924e-d59c-4340-9839-fbf25591be5c}
   Action UP01_Backbone_active: Id {46b55eec-8aa5-43cd-829a-7c4e25877f56} *)
